// TIA Portal project "Project2_22" (V15.1)

(* hardware
DEVICE "S7-1200 station_1"  S7-1200 Station
   slot 0: "Rack_0"  S7-1200 Rack  Rack  V1.0
   slot 1: "PLC_1"  CPU 1215C DC/DC/DC  6ES7 215-1AG40-0XB0  V4.3
*)

// ===== PLC "PLC_1"  CPU 1215C DC/DC/DC =====

VAR_GLOBAL   // PLC tag table "Default tag table"
   "porshen1" AT %Q1.0 : Bool;
   "porshen2" AT %Q0.7 : Bool;
   "snimac1" AT %I0.7 : Bool;
   "snimac2" AT %I0.2 : Bool;
   "KS1" AT %I1.0 : Bool;
   "KS2" AT %I0.6 : Bool;
   "dopravnik" AT %Q0.2 : Bool;
   "otocnik" AT %Q0.4 : Bool;
   "kompressor" AT %Q1.1 : Bool;
   "porshen3poz3" AT %Q0.5 : Bool;
   "porshen3poz5" AT %Q0.6 : Bool;
   "Tag_1" AT %M100.7 : Bool;
   "P" AT %M101.0 : Bool;
   "P3" AT %M101.1 : Bool;
   "pomocka_prosto_tak" AT %M101.2 : Bool;
   "PO" AT %M101.3 : Bool;
   "ppp" AT %M101.4 : Bool;
END_VAR

DATA_BLOCK "PIEST_DB1"   // DB1
{ S7_Optimized_Access := 'TRUE' }
VERSION : 0.1
// stored: InstanceOfName PIEST
"PIEST"
BEGIN
END_DATA_BLOCK

DATA_BLOCK "OS_DB"   // DB2
{ S7_Optimized_Access := 'TRUE' }
VERSION : 0.1
// stored: InstanceOfName OS
"OS"
BEGIN
END_DATA_BLOCK

DATA_BLOCK "PIEST_DB2"   // DB3
{ S7_Optimized_Access := 'TRUE' }
VERSION : 0.1
// stored: InstanceOfName PIEST
"PIEST"
BEGIN
END_DATA_BLOCK

DATA_BLOCK "PIEST_DB3"   // DB4
{ S7_Optimized_Access := 'TRUE' }
VERSION : 0.1
// stored: InstanceOfName PIEST
"PIEST"
BEGIN
END_DATA_BLOCK

DATA_BLOCK "DOPRAVNIK_FC_DB"   // DB5
{ S7_Optimized_Access := 'TRUE' }
VERSION : 0.1
// stored: InstanceOfName DOPRAVNIK_FC
"DOPRAVNIK_FC"
BEGIN
END_DATA_BLOCK

// folder: System blocks/Program resources

DATA_BLOCK "IEC_Timer_0_DB"   // DB6
{ S7_Optimized_Access := 'TRUE' }
AUTHOR : Simatic
FAMILY : IEC
NAME : IEC_TMR
VERSION : 1.0
// stored: InstanceOfName IEC_TIMER
"IEC_TIMER"
BEGIN
END_DATA_BLOCK

// folder: (top level)

FUNCTION_BLOCK "PIEST"   // FB1, LAD
{ S7_Optimized_Access := 'TRUE' }
VERSION : 0.1
   VAR_INPUT
      START : Bool;
      N : Int;
      pozastav : Bool;
      pozicia : Bool;
   END_VAR
   VAR_OUTPUT
      VZAD : Bool;
      PRED : Bool;
   END_VAR
   VAR
      HOTOVO : Bool;
      static1 : Bool;
      PRACUJEM : Bool;
   END_VAR
   VAR RETAIN
      IEC_Counter_0_Instance : CTU_INT;
   END_VAR
   VAR
      IEC_Timer_0_Instance : TON_TIME;
      IEC_Timer_0_Instance_1 : TON_TIME;
      IEC_Timer_0_Instance_2 : TON_TIME;
      IEC_Timer_0_Instance_3 : TON_TIME;
      IEC_Timer_0_Instance_4 : TON_TIME;
   END_VAR
   VAR_TEMP   // added for the SCL form of the ladder/FBD networks
      _w1 : Bool;
      _w2 : Bool;
   END_VAR
BEGIN

REGION Network 1
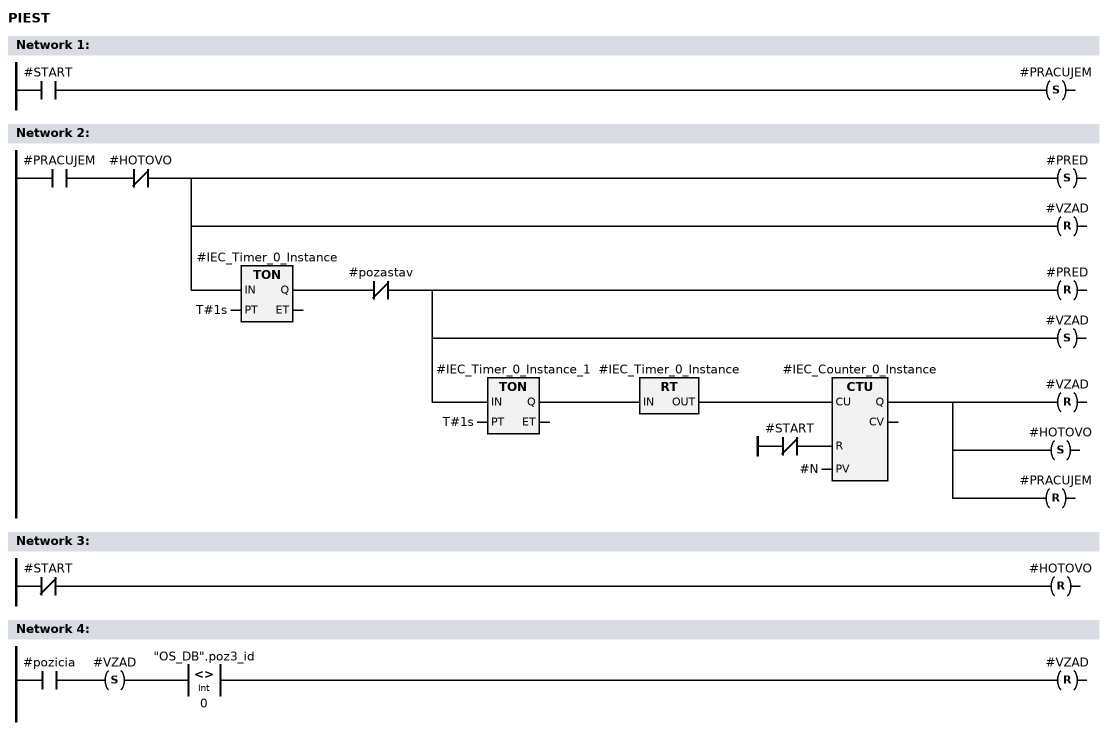
   RUNG wire#powerrail
      Contact( #START )
      S_Coil( #PRACUJEM )
   END_RUNG
   // the same network as SCL:
   IF #START THEN #PRACUJEM := TRUE; END_IF;
END_REGION

REGION Network 2
   #_w1 := #PRACUJEM AND NOT #HOTOVO;
   IF #_w1 THEN
       #PRED := TRUE;
       #VZAD := FALSE;
   END_IF;
   #IEC_Timer_0_Instance(IN := #_w1, PT := T#1s);   // TON
   #_w2 := #IEC_Timer_0_Instance.Q AND NOT #pozastav;
   IF #_w2 THEN
       #PRED := FALSE;
       #VZAD := TRUE;
   END_IF;
   #IEC_Timer_0_Instance_1(IN := #_w2, PT := T#1s);   // TON
   IF #IEC_Timer_0_Instance_1.Q THEN RESET_TIMER(#IEC_Timer_0_Instance); END_IF;
   #IEC_Counter_0_Instance(CU := #IEC_Timer_0_Instance_1.Q, R := NOT #START, PV := #N);   // CTU
   IF #IEC_Counter_0_Instance.Q THEN
       #VZAD := FALSE;
       #HOTOVO := TRUE;
       #PRACUJEM := FALSE;
   END_IF;
END_REGION

REGION Network 3
   RUNG wire#powerrail
      I_Contact( #START )
      R_Coil( #HOTOVO )
   END_RUNG
   // the same network as SCL:
   IF NOT #START THEN #HOTOVO := FALSE; END_IF;
END_REGION

REGION Network 4
   RUNG wire#powerrail
      Contact( #pozicia )
      S_Coil( #VZAD )
      { S7_Templates := "SrcType := Int" } NE_Contact(in1 := "OS_DB".poz3_id, in2 := 0)
      R_Coil( #VZAD )
   END_RUNG
   // the same network as SCL:
   IF #pozicia THEN #VZAD := TRUE; END_IF;
   IF #pozicia AND ("OS_DB".poz3_id <> 0) THEN #VZAD := FALSE; END_IF;
END_REGION
END_FUNCTION_BLOCK

FUNCTION_BLOCK "OS"   // FB2, LAD
{ S7_Optimized_Access := 'TRUE' }
VERSION : 0.1
   VAR_INPUT
      CISLO_IN : Int;
      NALOZENY : Bool;
      START : Bool;
      TL_IN : Bool;
      TL_OUT : Bool;
      PRAZDNA : Bool;
      EN_MOVEMENT : Bool;
      LOADED : Bool;
   END_VAR
   VAR_OUTPUT
      krytus : Bool;
   END_VAR
   VAR
      poz1_id : Int;
      poz2_id : Int;
      poz3_id : Int;
      poz4_id : Int;
      OK_POZICIA : Bool;
      IEC_Timer_0_Instance : TON_TIME;
      R_TRIG_Instance : R_TRIG;
      nechanivanie_id : Int;
   END_VAR
   VAR_TEMP   // added for the SCL form of the ladder/FBD networks
      _w1 : Bool;
   END_VAR
BEGIN

REGION Network 1
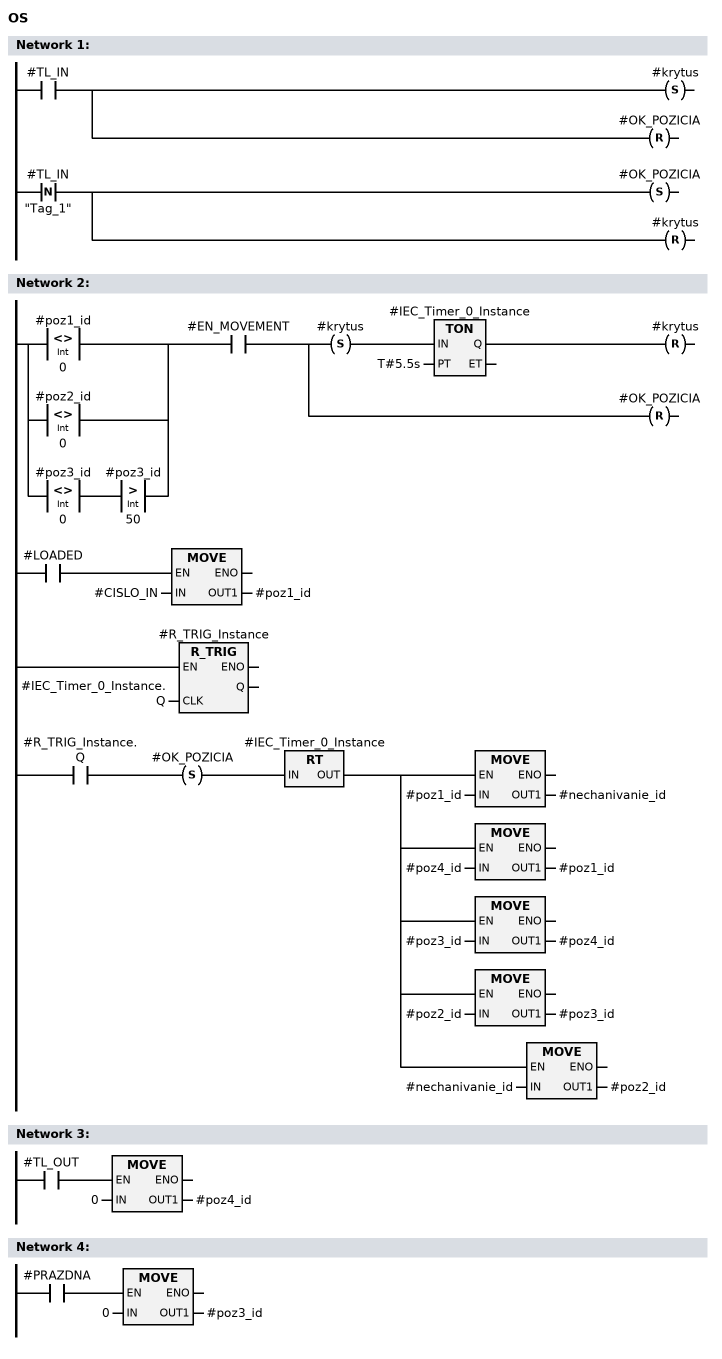
   RUNG wire#powerrail
      Contact( #TL_IN )
      wire#w1
      S_Coil( #krytus )
   END_RUNG
   RUNG wire#w1
      R_Coil( #OK_POZICIA )
   END_RUNG
   RUNG wire#powerrail
      N_Contact(operand := #TL_IN, bit := "Tag_1")
      wire#w2
      S_Coil( #OK_POZICIA )
   END_RUNG
   RUNG wire#w2
      R_Coil( #krytus )
   END_RUNG
   // the same network as SCL:
   IF #TL_IN THEN
       #krytus := TRUE;
       #OK_POZICIA := FALSE;
   END_IF;
   #_w1 := NOT #TL_IN AND "Tag_1";   // falling edge of #TL_IN
   "Tag_1" := #TL_IN;
   IF #_w1 THEN
       #OK_POZICIA := TRUE;
       #krytus := FALSE;
   END_IF;
END_REGION

REGION Network 2
   #_w1 := ((#poz1_id <> 0) OR (#poz2_id <> 0) OR ((#poz3_id <> 0) AND (#poz3_id > 50))) AND #EN_MOVEMENT;
   IF #_w1 THEN #krytus := TRUE; END_IF;
   #IEC_Timer_0_Instance(IN := #_w1, PT := T#5.5s);   // TON
   IF #IEC_Timer_0_Instance.Q THEN #krytus := FALSE; END_IF;
   IF #_w1 THEN #OK_POZICIA := FALSE; END_IF;
   IF #LOADED THEN #poz1_id := #CISLO_IN; END_IF;
   #R_TRIG_Instance(CLK := #IEC_Timer_0_Instance.Q);   // R_TRIG
   IF #R_TRIG_Instance.Q THEN
       #OK_POZICIA := TRUE;
       RESET_TIMER(#IEC_Timer_0_Instance);
       #nechanivanie_id := #poz1_id;
       #poz1_id := #poz4_id;
       #poz4_id := #poz3_id;
       #poz3_id := #poz2_id;
       #poz2_id := #nechanivanie_id;
   END_IF;
END_REGION

REGION Network 3
   RUNG wire#powerrail
      Contact( #TL_OUT )
      Move(in := 0, out1 => #poz4_id)
   END_RUNG
   // the same network as SCL:
   IF #TL_OUT THEN #poz4_id := 0; END_IF;
END_REGION

REGION Network 4
   RUNG wire#powerrail
      Contact( #PRAZDNA )
      Move(in := 0, out1 => #poz3_id)
   END_RUNG
   // the same network as SCL:
   IF #PRAZDNA THEN #poz3_id := 0; END_IF;
END_REGION
END_FUNCTION_BLOCK

FUNCTION_BLOCK "DOPRAVNIK_FC"   // FB3, LAD
{ S7_Optimized_Access := 'TRUE' }
VERSION : 0.1
   VAR_INPUT
      START : Bool;
      STOP : Bool;
      LOADED : Bool;
      CISLO_IN : Int;
   END_VAR
   VAR_OUTPUT
      MOVE : Bool;
   END_VAR
   VAR
      PRACUJEM : Bool;
      Static_1 : Bool;
      Static_2 : Bool;
      Static_3 : Bool;
      poz5_id : Int;
      poz6_id : Int;
      IEC_Timer_0_Instance : TON_TIME;
      IEC_Timer_0_Instance_1 : TON_TIME;
      IEC_Timer_0_Instance_2 : TON_TIME;
      IEC_Timer_0_Instance_3 : TON_TIME;
      IEC_Timer_0_Instance_4 : TON_TIME;
      IEC_Timer_0_Instance_5 : TON_TIME;
   END_VAR
   VAR_TEMP
      nechavanie : Int;
   END_VAR
   VAR_TEMP   // added for the SCL form of the ladder/FBD networks
      _w1 : Bool;
      _w2 : Bool;
   END_VAR
BEGIN

REGION Network 1
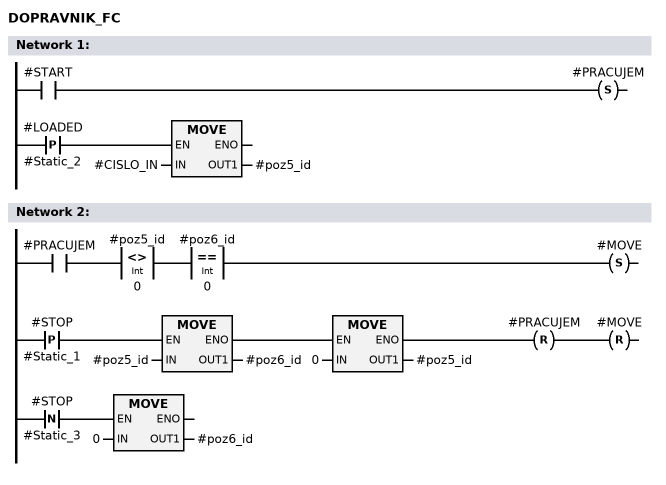
   RUNG wire#powerrail
      Contact( #START )
      S_Coil( #PRACUJEM )
   END_RUNG
   RUNG wire#powerrail
      P_Contact(operand := #LOADED, bit := #Static_2)
      Move(in := #CISLO_IN, out1 => #poz5_id)
   END_RUNG
   // the same network as SCL:
   IF #START THEN #PRACUJEM := TRUE; END_IF;
   #_w1 := #LOADED AND NOT #Static_2;   // rising edge of #LOADED
   #Static_2 := #LOADED;
   IF #_w1 THEN #poz5_id := #CISLO_IN; END_IF;
END_REGION

REGION Network 2
   RUNG wire#powerrail
      Contact( #PRACUJEM )
      { S7_Templates := "SrcType := Int" } NE_Contact(in1 := #poz5_id, in2 := 0)
      { S7_Templates := "SrcType := Int" } EQ_Contact(in1 := #poz6_id, in2 := 0)
      S_Coil( #MOVE )
   END_RUNG
   RUNG wire#powerrail
      P_Contact(operand := #STOP, bit := #Static_1)
      Move(in := #poz5_id, out1 => #poz6_id)
      Move(in := 0, out1 => #poz5_id)
      R_Coil( #PRACUJEM )
      R_Coil( #MOVE )
   END_RUNG
   RUNG wire#powerrail
      N_Contact(operand := #STOP, bit := #Static_3)
      Move(in := 0, out1 => #poz6_id)
   END_RUNG
   // the same network as SCL:
   IF #PRACUJEM AND (#poz5_id <> 0) AND (#poz6_id = 0) THEN #MOVE := TRUE; END_IF;
   #_w1 := #STOP AND NOT #Static_1;   // rising edge of #STOP
   #Static_1 := #STOP;
   IF #_w1 THEN
       #poz6_id := #poz5_id;
       #poz5_id := 0;
       #PRACUJEM := FALSE;
       #MOVE := FALSE;
   END_IF;
   #_w2 := NOT #STOP AND #Static_3;   // falling edge of #STOP
   #Static_3 := #STOP;
   IF #_w2 THEN #poz6_id := 0; END_IF;
END_REGION
END_FUNCTION_BLOCK

ORGANIZATION_BLOCK "Main"   // OB1, LAD, ProgramCycle
TITLE = "Main Program Sweep (Cycle)"
{ S7_Optimized_Access := 'TRUE' }
VERSION : 0.1
   VAR_INPUT
      Initial_Call : Bool;   // Initial call of this OB
      Remanence : Bool;   // =True, if remanent data are available
   END_VAR
BEGIN

REGION Network 1: os
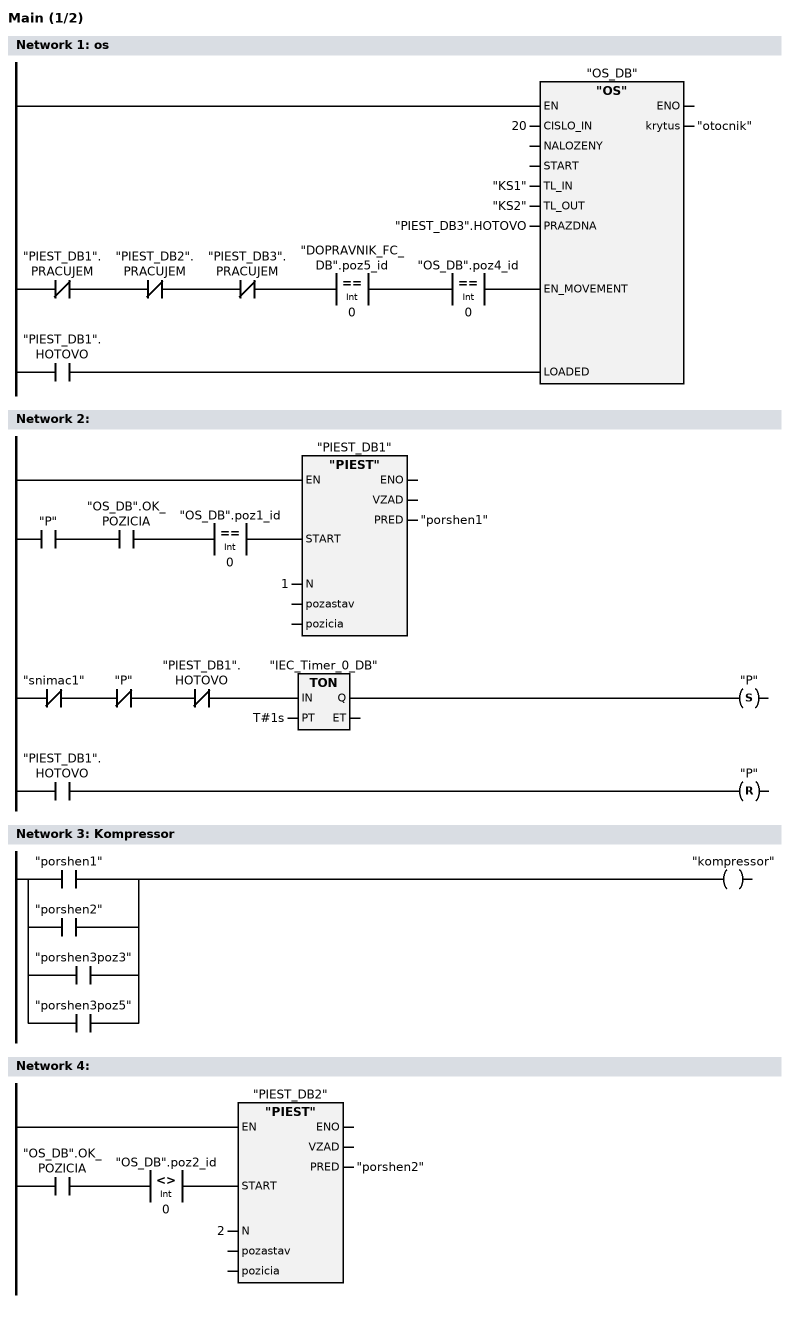
   RUNG wire#powerrail
      "OS_DB"(EN_MOVEMENT := wire#w1, LOADED := wire#w2, CISLO_IN := 20, NALOZENY :=, START :=, TL_IN := "KS1", TL_OUT := "KS2", PRAZDNA := "PIEST_DB3".HOTOVO, krytus => "otocnik")
   END_RUNG
   RUNG wire#powerrail
      I_Contact( "PIEST_DB1".PRACUJEM )
      I_Contact( "PIEST_DB2".PRACUJEM )
      I_Contact( "PIEST_DB3".PRACUJEM )
      { S7_Templates := "SrcType := Int" } EQ_Contact(in1 := "DOPRAVNIK_FC_DB".poz5_id, in2 := 0)
      { S7_Templates := "SrcType := Int" } EQ_Contact(in1 := "OS_DB".poz4_id, in2 := 0)
   END_RUNG wire#w1
   RUNG wire#powerrail
      Contact( "PIEST_DB1".HOTOVO )
   END_RUNG wire#w2
   // the same network as SCL:
   "OS_DB"(CISLO_IN := 20,   // "OS"
           TL_IN := "KS1",
           TL_OUT := "KS2",
           PRAZDNA := "PIEST_DB3".HOTOVO,
           EN_MOVEMENT := NOT "PIEST_DB1".PRACUJEM AND NOT "PIEST_DB2".PRACUJEM AND NOT "PIEST_DB3".PRACUJEM AND ("DOPRAVNIK_FC_DB".poz5_id = 0) AND ("OS_DB".poz4_id = 0),
           LOADED := "PIEST_DB1".HOTOVO,
           krytus => "otocnik");
END_REGION

REGION Network 2
   "PIEST_DB1"(START := "P" AND "OS_DB".OK_POZICIA AND ("OS_DB".poz1_id = 0), N := 1, PRED => "porshen1");   // "PIEST"
   "IEC_Timer_0_DB".TON(IN := NOT "snimac1" AND NOT "P" AND NOT "PIEST_DB1".HOTOVO, PT := T#1s);
   IF "IEC_Timer_0_DB".Q THEN "P" := TRUE; END_IF;
   IF "PIEST_DB1".HOTOVO THEN "P" := FALSE; END_IF;
END_REGION

REGION Network 3: Kompressor
   RUNG wire#powerrail
      Contact( "porshen1" )
      wire#w1
      Coil( "kompressor" )
   END_RUNG
   RUNG wire#powerrail
      Contact( "porshen2" )
   END_RUNG wire#w1
   RUNG wire#powerrail
      Contact( "porshen3poz3" )
   END_RUNG wire#w1
   RUNG wire#powerrail
      Contact( "porshen3poz5" )
   END_RUNG wire#w1
   // the same network as SCL:
   "kompressor" := "porshen1" OR "porshen2" OR "porshen3poz3" OR "porshen3poz5";
END_REGION

REGION Network 4
   RUNG wire#powerrail
      "PIEST_DB2"(START := wire#w1, N := 2, pozastav :=, pozicia :=, VZAD =>, PRED => "porshen2")
   END_RUNG
   RUNG wire#powerrail
      Contact( "OS_DB".OK_POZICIA )
      { S7_Templates := "SrcType := Int" } NE_Contact(in1 := "OS_DB".poz2_id, in2 := 0)
   END_RUNG wire#w1
   // the same network as SCL:
   "PIEST_DB2"(START := "OS_DB".OK_POZICIA AND ("OS_DB".poz2_id <> 0), N := 2, PRED => "porshen2");   // "PIEST"
END_REGION

REGION Network 5
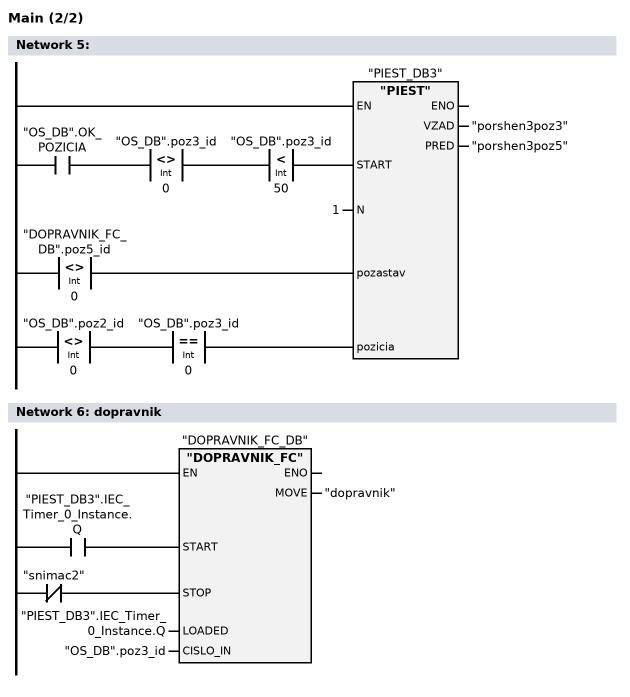
   RUNG wire#powerrail
      "PIEST_DB3"(START := wire#w1, pozastav := wire#w2, pozicia := wire#w3, N := 1, VZAD => "porshen3poz3", PRED => "porshen3poz5")
   END_RUNG
   RUNG wire#powerrail
      Contact( "OS_DB".OK_POZICIA )
      { S7_Templates := "SrcType := Int" } NE_Contact(in1 := "OS_DB".poz3_id, in2 := 0)
      { S7_Templates := "SrcType := Int" } LT_Contact(in1 := "OS_DB".poz3_id, in2 := 50)
   END_RUNG wire#w1
   RUNG wire#powerrail
      { S7_Templates := "SrcType := Int" } NE_Contact(in1 := "DOPRAVNIK_FC_DB".poz5_id, in2 := 0)
   END_RUNG wire#w2
   RUNG wire#powerrail
      { S7_Templates := "SrcType := Int" } NE_Contact(in1 := "OS_DB".poz2_id, in2 := 0)
      { S7_Templates := "SrcType := Int" } EQ_Contact(in1 := "OS_DB".poz3_id, in2 := 0)
   END_RUNG wire#w3
   // the same network as SCL:
   "PIEST_DB3"(START := "OS_DB".OK_POZICIA AND ("OS_DB".poz3_id <> 0) AND ("OS_DB".poz3_id < 50),   // "PIEST"
               N := 1,
               pozastav := "DOPRAVNIK_FC_DB".poz5_id <> 0,
               pozicia := ("OS_DB".poz2_id <> 0) AND ("OS_DB".poz3_id = 0),
               VZAD => "porshen3poz3",
               PRED => "porshen3poz5");
END_REGION

REGION Network 6: dopravnik
   RUNG wire#powerrail
      "DOPRAVNIK_FC_DB"(START := wire#w1, STOP := wire#w2, LOADED := "PIEST_DB3".IEC_Timer_0_Instance.Q, CISLO_IN := "OS_DB".poz3_id, MOVE => "dopravnik")
   END_RUNG
   RUNG wire#powerrail
      Contact( "PIEST_DB3".IEC_Timer_0_Instance.Q )
   END_RUNG wire#w1
   RUNG wire#powerrail
      I_Contact( "snimac2" )
   END_RUNG wire#w2
   // the same network as SCL:
   "DOPRAVNIK_FC_DB"(START := "PIEST_DB3".IEC_Timer_0_Instance.Q,   // "DOPRAVNIK_FC"
                     STOP := NOT "snimac2",
                     LOADED := "PIEST_DB3".IEC_Timer_0_Instance.Q,
                     CISLO_IN := "OS_DB".poz3_id,
                     MOVE => "dopravnik");
END_REGION
END_ORGANIZATION_BLOCK